# EPICS substitutions: iocBoot/ioc13bma_linux/auto_shutter.substitutions
file "$(CARS)/db/auto_shutter.db"
{
pattern
{P,      SHUT, SHUT_STATUS,       SHUT_CONTROL,        PERIOD, BEAM_READY}
{13BMA:, FOE,  13BMA:eps_mbbi4,   13BMA:OpenFEShutter,  30,    PA:13BM:STA_A_BEAMREADY_PL}
{13BMA:, BMC,  13BMA:eps_mbbi100, 13BMA:OpenBMCShutter, 30,    PA:13BM:STA_C_BEAMREADY_PL}
{13BMA:, BMD,  13BMA:eps_mbbi99,  13BMA:OpenBMDShutter, 30,    PA:13BM:STA_D_BEAMREADY_PL}
}
